	Bypass: BOOL;
	bogus: BOOL := FALSE;
	SR_FD2_new: SR;
	fbWasteBlower: TOF;
	
	bHotMeltAlarm_i:BOOL;
	
END_VAR

VAR_OUTPUT
	bHighHeatOn_i: BOOL;
	bBlowerOn_i: BOOL;
END_VAR

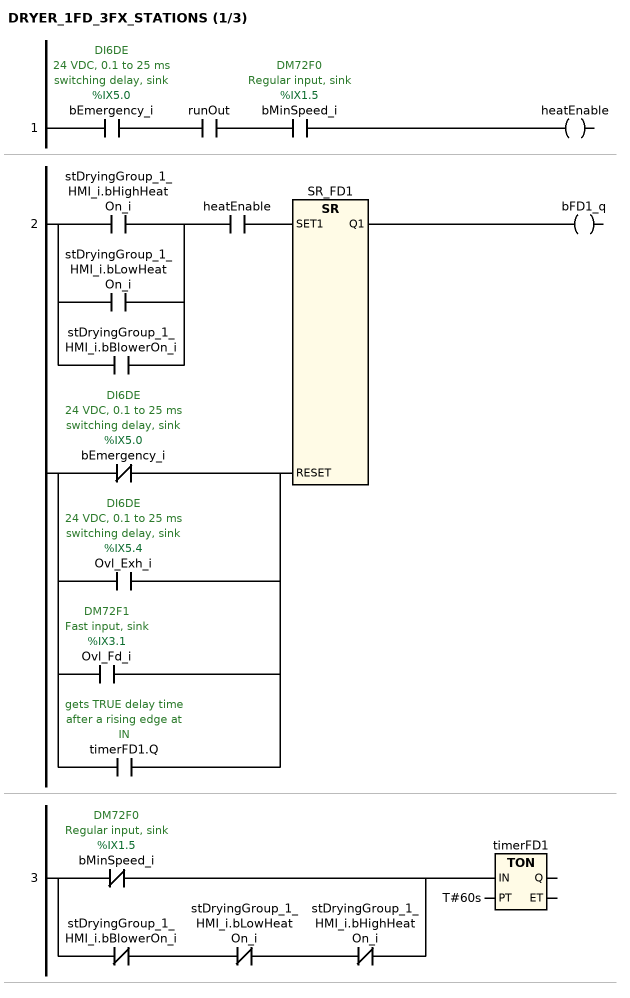
// NETWORK 1
//   bEmergency_i: DI6DE 24 VDC, 0.1 to 25 ms switching delay, sink | AT %IX5.0
//   bMinSpeed_i: DM72F0 Regular input, sink | AT %IX1.5
heatEnable := bEmergency_i AND runOut AND bMinSpeed_i;

// NETWORK 2
//   bEmergency_i: DI6DE 24 VDC, 0.1 to 25 ms switching delay, sink | AT %IX5.0
//   Ovl_Exh_i: DI6DE 24 VDC, 0.1 to 25 ms switching delay, sink | AT %IX5.4
//   Ovl_Fd_i: DM72F1 Fast input, sink | AT %IX3.1
//   timerFD1.Q: gets TRUE delay time after a rising edge at IN
SR_FD1(SET1 := (stDryingGroup_1_HMI_i.bHighHeatOn_i OR stDryingGroup_1_HMI_i.bLowHeatOn_i OR stDryingGroup_1_HMI_i.bBlowerOn_i) AND heatEnable, RESET := NOT bEmergency_i OR Ovl_Exh_i OR Ovl_Fd_i OR timerFD1.Q); // SR
bFD1_q := SR_FD1.Q1;

// NETWORK 3
//   bMinSpeed_i: DM72F0 Regular input, sink | AT %IX1.5
timerFD1(IN := NOT bMinSpeed_i OR NOT stDryingGroup_1_HMI_i.bBlowerOn_i AND NOT stDryingGroup_1_HMI_i.bLowHeatOn_i AND NOT stDryingGroup_1_HMI_i.bHighHeatOn_i, PT := T#60s); // TON

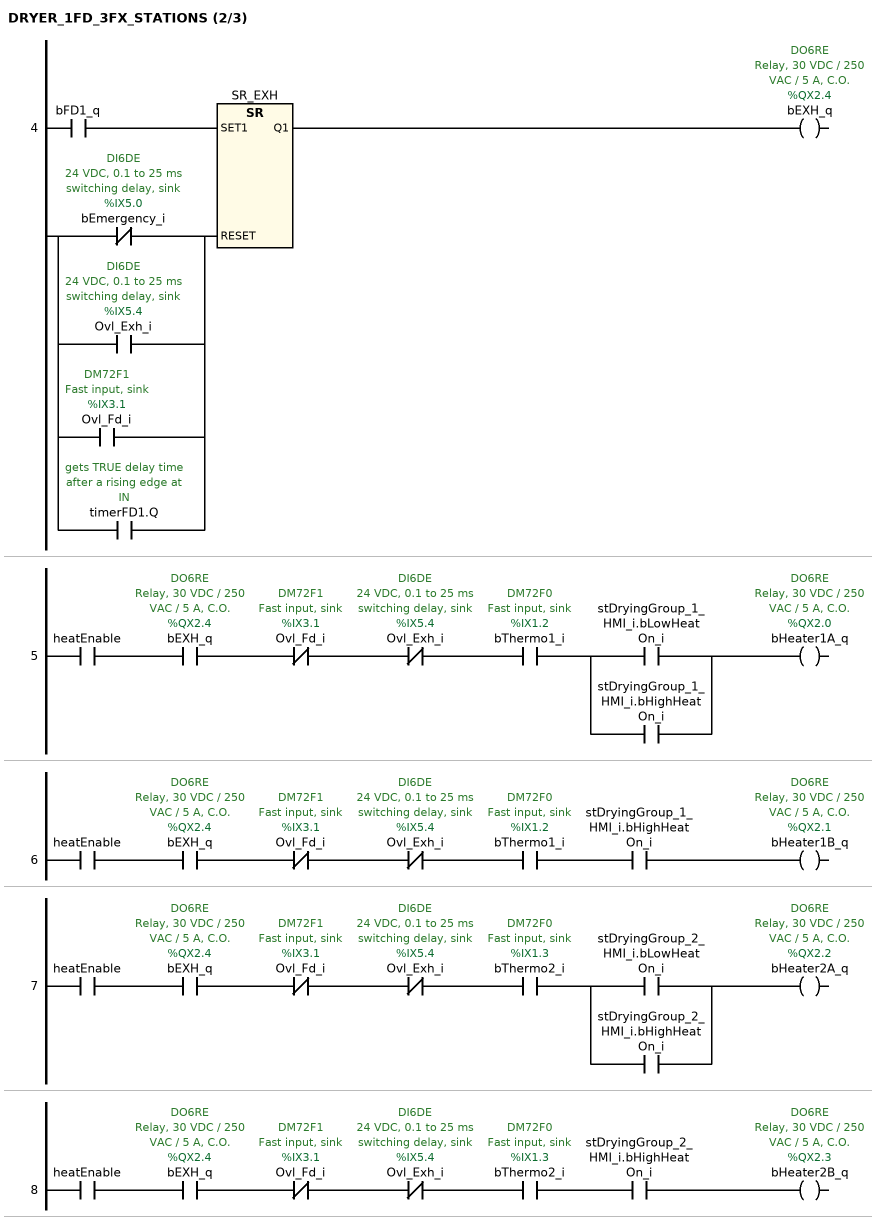
// NETWORK 4
//   bEmergency_i: DI6DE 24 VDC, 0.1 to 25 ms switching delay, sink | AT %IX5.0
//   Ovl_Exh_i: DI6DE 24 VDC, 0.1 to 25 ms switching delay, sink | AT %IX5.4
//   Ovl_Fd_i: DM72F1 Fast input, sink | AT %IX3.1
//   timerFD1.Q: gets TRUE delay time after a rising edge at IN
//   bEXH_q: DO6RE Relay, 30 VDC / 250 VAC / 5 A, C.O. | AT %QX2.4
SR_EXH(SET1 := bFD1_q, RESET := NOT bEmergency_i OR Ovl_Exh_i OR Ovl_Fd_i OR timerFD1.Q); // SR
bEXH_q := SR_EXH.Q1;

// NETWORK 5
//   bEXH_q: DO6RE Relay, 30 VDC / 250 VAC / 5 A, C.O. | AT %QX2.4
//   Ovl_Fd_i: DM72F1 Fast input, sink | AT %IX3.1
//   Ovl_Exh_i: DI6DE 24 VDC, 0.1 to 25 ms switching delay, sink | AT %IX5.4
//   bThermo1_i: DM72F0 Fast input, sink | AT %IX1.2
//   bHeater1A_q: DO6RE Relay, 30 VDC / 250 VAC / 5 A, C.O. | AT %QX2.0
bHeater1A_q := heatEnable AND bEXH_q AND NOT Ovl_Fd_i AND NOT Ovl_Exh_i AND bThermo1_i AND (stDryingGroup_1_HMI_i.bLowHeatOn_i OR stDryingGroup_1_HMI_i.bHighHeatOn_i);

// NETWORK 6
//   bEXH_q: DO6RE Relay, 30 VDC / 250 VAC / 5 A, C.O. | AT %QX2.4
//   Ovl_Fd_i: DM72F1 Fast input, sink | AT %IX3.1
//   Ovl_Exh_i: DI6DE 24 VDC, 0.1 to 25 ms switching delay, sink | AT %IX5.4
//   bThermo1_i: DM72F0 Fast input, sink | AT %IX1.2
//   bHeater1B_q: DO6RE Relay, 30 VDC / 250 VAC / 5 A, C.O. | AT %QX2.1
bHeater1B_q := heatEnable AND bEXH_q AND NOT Ovl_Fd_i AND NOT Ovl_Exh_i AND bThermo1_i AND stDryingGroup_1_HMI_i.bHighHeatOn_i;

// NETWORK 7
//   bEXH_q: DO6RE Relay, 30 VDC / 250 VAC / 5 A, C.O. | AT %QX2.4
//   Ovl_Fd_i: DM72F1 Fast input, sink | AT %IX3.1
//   Ovl_Exh_i: DI6DE 24 VDC, 0.1 to 25 ms switching delay, sink | AT %IX5.4
//   bThermo2_i: DM72F0 Fast input, sink | AT %IX1.3
//   bHeater2A_q: DO6RE Relay, 30 VDC / 250 VAC / 5 A, C.O. | AT %QX2.2
bHeater2A_q := heatEnable AND bEXH_q AND NOT Ovl_Fd_i AND NOT Ovl_Exh_i AND bThermo2_i AND (stDryingGroup_2_HMI_i.bLowHeatOn_i OR stDryingGroup_2_HMI_i.bHighHeatOn_i);

// NETWORK 8
//   bEXH_q: DO6RE Relay, 30 VDC / 250 VAC / 5 A, C.O. | AT %QX2.4
//   Ovl_Fd_i: DM72F1 Fast input, sink | AT %IX3.1
//   Ovl_Exh_i: DI6DE 24 VDC, 0.1 to 25 ms switching delay, sink | AT %IX5.4
//   bThermo2_i: DM72F0 Fast input, sink | AT %IX1.3
//   bHeater2B_q: DO6RE Relay, 30 VDC / 250 VAC / 5 A, C.O. | AT %QX2.3
bHeater2B_q := heatEnable AND bEXH_q AND NOT Ovl_Fd_i AND NOT Ovl_Exh_i AND bThermo2_i AND stDryingGroup_2_HMI_i.bHighHeatOn_i;

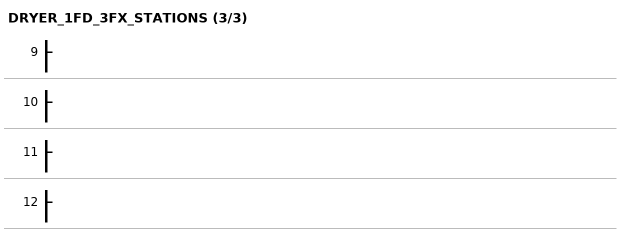
// NETWORK 9

// NETWORK 10

// NETWORK 11

// NETWORK 12

END_PROGRAM

// MyController/Application/ETH_NETWORK
PROGRAM ETH_NETWORK
VAR
	

	NewWord: WORD;
	NewBool:	BOOL;
	
	ReINIT:BOOL := FALSE;
	bTest_MinSpeed_i:BOOL := FALSE;
	
	
	FromRewind:WORD	:=	0;
	fbTP_STARTUP: TP;
	tStartUp_Time:TIME;
	AniloxModbusError2: BOOL;
	
	RexrothModbusError: BOOL;
	
	FB_RegPos: TP;
	FB_RegNeg: TP;
	
	FB_JogPos: TP;
	FB_JogNeg: TP;
END_VAR




bStartUpBit	:= TRUE;
fbTP_STARTUP(IN:=bStartUpBit , PT:= T#3S, Q=> bStartUp_ResetBit, ET=> tStartUp_Time);
fbTP_STARTUP(IN:=bStartUpBit , PT:= T#3S, Q=> bStartUp_SetBit, ET=> tStartUp_Time);

IF bStartUp_SetBit = TRUE AND uiUnwindTensManual_HMI_i = 0 THEN
	
	uiUnwindTensManual_HMI_i:= 10;
END_IF


wPar1838_PidOn_ETH.0 := bRewindPID_Out; 
InfeedModbusError	:= IoConfig_Globals.INFEED_Instance.xError;


IF InfeedModbusError = TRUE THEN

	
	IoConfig_Globals.INFEED_Instance.xConfirmError := TRUE;

ELSE		
	IoConfig_Globals.INFEED_Instance.xConfirmError := FALSE;
END_IF



RewindModbusError	:= IoConfig_Globals.REWIND_DF_Instance.xError;


IF RewindModbusError = TRUE THEN

	IoConfig_Globals.REWIND_DF_Instance.xConfirmError := TRUE;

ELSE		
	IoConfig_Globals.REWIND_DF_Instance.xConfirmError := FALSE;
END_IF


// TOP REWIND COMM ERROR MANAGE
TopRewindModbusError	:= IoConfig_Globals.TOP_REWIND_Instance.xError;

IF TopRewindModbusError = TRUE THEN

	
	IoConfig_Globals.TOP_REWIND_Instance.xConfirmError := TRUE;

ELSE		
	IoConfig_Globals.TOP_REWIND_Instance.xConfirmError := FALSE;
END_IF



// GRAVURE COMM ERROR MANAGE
GravureModbusError	:= IoConfig_Globals.GRAVURE_Instance.xError;

IF GravureModbusError = TRUE THEN

	
	IoConfig_Globals.GRAVURE_Instance.xConfirmError := TRUE;

ELSE		
	IoConfig_Globals.GRAVURE_Instance.xConfirmError := FALSE;
END_IF


IF gravureOnOut = TRUE THEN
	
//wRexrothCmd.0;
NewBool:= TRUE;
ELSE
NewBool:= FALSE;
//wRexrothCmd.0;

END_IF


//ANILOX COMM ERROR MANAGE

AniloxModbusError	:= IoConfig_Globals.ANILOX_1_Instance.xError;
//IoConfig_Globals.REWIND_Instance.xConfirmError := ReINIT;

IF AniloxModbusError = TRUE THEN

	IoConfig_Globals.ANILOX_1_Instance.xConfirmError := TRUE;

ELSE		
	IoConfig_Globals.ANILOX_1_Instance.xConfirmError := FALSE;
END_IF


AniloxModbusError2	:= IoConfig_Globals.ANILOX_2_Instance.xError;
//IoConfig_Globals.REWIND_Instance.xConfirmError := ReINIT;

IF AniloxModbusError2 = TRUE THEN

	IoConfig_Globals.ANILOX_2_Instance.xConfirmError := TRUE;

ELSE		
	IoConfig_Globals.ANILOX_2_Instance.xConfirmError := FALSE;
END_IF

IF infeedOnOut = TRUE THEN
	
	wPar1837_InfeedOn_ETH	:= 1;
ELSE
	wPar1837_InfeedOn_ETH	:= 0;

END_IF


IF bGravureRegiOn_HMI_q = TRUE THEN
	
	wPar1838_FilterOn_ETH	:= 1;
ELSE
	wPar1838_FilterOn_ETH	:= 0;

END_IF



//REWIND ON / OFF
IF (rewindOnOut = TRUE ) THEN
	
	wPar1837_RewindOn_ETH	:= 1;
ELSE
	wPar1837_RewindOn_ETH	:= 0;
	
END_IF


//REWIND PID ON
IF bRewindPID_Out = TRUE THEN
	
	wPar1838_PidOn_ETH	:= 1;
	
ELSE
	wPar1838_PidOn_ETH	:= 0;

	
END_IF



//TOP REWIND ON / OFF
IF GVL_HMI.top_rewindOnOut  = TRUE THEN
	

	wPar1837_TopRewindOn_ETH	:= 1;
ELSE
	wPar1837_TopRewindOn_ETH	:= 0;
	
END_IF


//TOP REWIND PID ON  (SAME SIGNAL)
IF bRewindPID_Out = TRUE THEN
	
	wPar1838_TopPidOn_ETH	:= 1;
	
ELSE
	wPar1838_TopPidOn_ETH	:= 0;

	
END_IF

//TOP REWIND ON / OFF
IF GVL_HMI.gravureOnOut  = TRUE THEN
	

	wPar1837_GravureOn_ETH	:= 1;
ELSE
	wPar1837_GravureOn_ETH	:= 0;
	
END_IF



IF ArFlexoStation[1].bAniloxMot_q = TRUE THEN
	
	wPar1838_ProcessOn_ETH := 0;	//ANILOX
ELSE
	wPar1838_ProcessOn_ETH := 1;	//ANILOX
END_IF

IF ArFlexoStation[2].bAniloxMot_q = TRUE THEN
	
	wPar1838_ProcessOn_2_ETH := 0;	//ANILOX
ELSE
	wPar1838_ProcessOn_2_ETH := 1;	//ANILOX
END_IF

wPar1839_AniloxFWD_ETH.0 	:= recto1Out;
wPar1840_AniloxBCK_ETH.0	:=	verso1Out;


wPar1839_AniloxFWD_2_ETH.0 	:= recto2Out;
wPar1840_AniloxBCK_2_ETH.0	:=	verso2Out;


IF (wPar2019_DryPermit_ETH.0) = TRUE THEN
	
	bTest_MinSpeed_i	:= 1;
ELSE
	bTest_MinSpeed_i	:= 0;
	
END_IF


IF (	(bArAniloxMotor_KEEP[1]) = TRUE) AND (NOT bArSETUP_KEEP[1]) THEN	


	wPar1837_AniloxOn_ETH	:= 1;
ELSE
	wPar1837_AniloxOn_ETH	:= 0;
	
END_IF


IF (	(bArAniloxMotor_KEEP[2]) = TRUE) AND (NOT bArSETUP_KEEP[2]) THEN	


	wPar1837_AniloxOn_2_ETH	:= 1;
ELSE
	wPar1837_AniloxOn_2_ETH	:= 0;
	
END_IF




IF (rollendOnOut = FALSE) THEN

	uiRollEndState := 0 ;
	
ELSIF ((rollendOnOut = TRUE) AND (bEndOfRoll_Reached = FALSE)) THEN

	uiRollEndState := 1 ;
	
ELSIF ((rollendOnOut = TRUE) AND (bEndOfRoll_Reached = TRUE)) THEN
	
	uiRollEndState := 2 ;
	
END_IF


bRewindHealthy_ETH := wPar1001_RewindHealthy_ETH.0;

bRewindActive_ETH	:= wPar1002_RewindActive_ETH.0;

bTopRewindHealthy_ETH := wPar1001_TopRewindHealthy_ETH.0;

bTopRewindActive_ETH	:= wPar1002_TopRewindActive_ETH.0;

bInfeedHealthy_ETH := 1;//wPar1001_InfeedHealthy_ETH.0;

bInfeedActive_ETH	:=  1;//wPar1002_InfeedActive_ETH.0;

IF ((bRewindHealthy_ETH AND bRewindActive_ETH) OR ( bConveyorOn_HMI_i) OR  (bTopRewindHealthy_ETH AND bTopRewindActive_ETH)) AND bInfeedHealthy_ETH AND bInfeedActive_ETH THEN
	
	bAllDrivesOK_TO_RUN_ETH := TRUE;
ELSE
	bAllDrivesOK_TO_RUN_ETH := FALSE;
	
END_IF

IF (bRewindHealthy_ETH AND bRewindActive_ETH) OR (bTopRewindHealthy_ETH AND bTopRewindActive_ETH) OR ( bConveyorOn_HMI_i) THEN

	bRewindRunSignalMissing_HMI := FALSE;
ELSE
	bRewindRunSignalMissing_HMI	:= TRUE;
END_IF

IF bInfeedHealthy_ETH AND bInfeedActive_ETH THEN

	bInfeedRunSignalMissing_HMI := FALSE;
ELSE
	bInfeedRunSignalMissing_HMI	:= TRUE;
END_IF


IF InfeedModbusError = TRUE OR RewindModbusError = TRUE  THEN
	
	bAllDrives_ModbusError_HMI := TRUE;
ELSE
	bAllDrives_ModbusError_HMI := FALSE;

END_IF

//****************************************
//*** GRAVURE COMMUNICATION MANAGEMENT ***
//****************************************

IoConfig_Globals.REXROTH_1_Instance.xBusy;
IoConfig_Globals.REXROTH_1_Instance.xError;
IoConfig_Globals.REXROTH_1_Instance.xDone;

// GRAVURE COMM ERROR MANAGE
RexrothModbusError	:= IoConfig_Globals.REXROTH_1_Instance.xError;

IF RexrothModbusError = TRUE THEN

	IoConfig_Globals.REXROTH_1_Instance.xConfirmError 	:= TRUE;
	
ELSE

	IoConfig_Globals.REXROTH_1_Instance.xConfirmError 	:= FALSE;

END_IF

	//IoConfig_Globals.REXROTH_1_Instance.x


bCounterReached_HMI_q := wPar1933_CountReach_ETH.0;

bGravure_Tens_Inc_ETH_q	:= bGravure_Tens_Inc_HMI_i;
bGravure_Tens_Dec_ETH_q	:= bGravure_Tens_Dec_HMI_i;
//bGravure_Tens_Inc_i	:= bGravure_Tens_Inc_HMI_i;
//bGravure_Tens_Dec_i	:= bGravure_Tens_Dec_HMI_i;
FB_RegPos(IN:=bGravure_Reg_Adv_HMI_i OR ArFlexoStation[1].bRegAdvance_q , PT:=T#250MS , Q=> , ET=> );
FB_RegNeg(IN:=bGravure_Reg_Ret_HMI_i OR ArFlexoStation[1].bRegRetard_q , PT:=T#250MS , Q=> , ET=> );

	bGravure_Reg_Adv_ETH_q	:= FB_RegPos.Q;
	bGravure_Reg_Ret_ETH_q	:= FB_RegNeg.Q;
	bGravureOn_ETH_q		:=	gravureOnOut;

	
	bGravureRegiOn_HMI_q		:=	bGravure_RegiCtrlOn_HMI_i;
	bInfeedRegiOn_HMI_q			:=	bInfeed_RegiCtrlOn_HMI_i;
	
FB_JogPos(IN:=bGravure_Jog_Adv_HMI_i , PT:=T#250MS , Q=> , ET=> );
FB_JogNeg(IN:=bGravure_Jog_Ret_HMI_i , PT:=T#250MS , Q=> , ET=> );

	bGravure_Jog_Adv_HMI_q		:=	FB_JogPos.Q;
	bGravure_Jog_Ret_HMI_q		:=	FB_JogNeg.Q;
	
//uiGravureRegisterOffset := WORD_TO_UINT(wGravureRegisterOffset);
uiGravureGearingAdjust := WORD_TO_UINT(wGravureGearingAdjust);

bInfeed_Tens_Inc_ETH_i := bInfeed_Tens_Inc_HMI_i;
bInfeed_Tens_dec_ETH_i :=bInfeed_Tens_dec_HMI_i;
bInfeed_Manual_ETH_i := bInfeed_Manual_i;
bInfeed_StatusError_HMI_q := bInfeed_StatusError_ETH_q;
bInfeed_StatusDisabled_q := ( NOT(bInfeed_StatusError_ETH_q) AND NOT  (bInfeed_StatusSynch_ETH_q) AND NOT  (bInfeed_StatusSlowRot_ETH_q));
bInfeed_StatusSynch_HMI_q :=bInfeed_StatusSynch_ETH_q;
bInfeed_ResetDrive_ETH_i := bInfeed_ResetDrive_HMI_i;

END_PROGRAM

// MyController/Application/FAULT_INTERLOCK
PROGRAM FAULT_INTERLOCK
VAR
	bogus: BOOL;
	SR_AniloxOn:		SR;
	bMachineHealthy:BOOL;
	
	
	infeedOnOut_L:BOOL;
	rewindOnOut_L:BOOL;
	
	bBYPASS:BOOL:= TRUE;
	
	okToRunV2:BOOL;
	okToJogV2:BOOL;
	fbTOF_RUN: TOF;
	etRun: TIME;
	bReadyToRun: BOOL;
	bSensorsOk: BOOL;
	SR_SlowRotation: SR;
	COUNTER_REACHED: BOOL;
END_VAR
VAR // added by the converter: edge detectors and wires of the graphical bodies
    _rt1, _rt2, _rt3, _rt4, _rt5, _rt6, _rt7, _rt8, _rt9, _rt10, _rt11, _rt12 : R_TRIG;
END_VAR

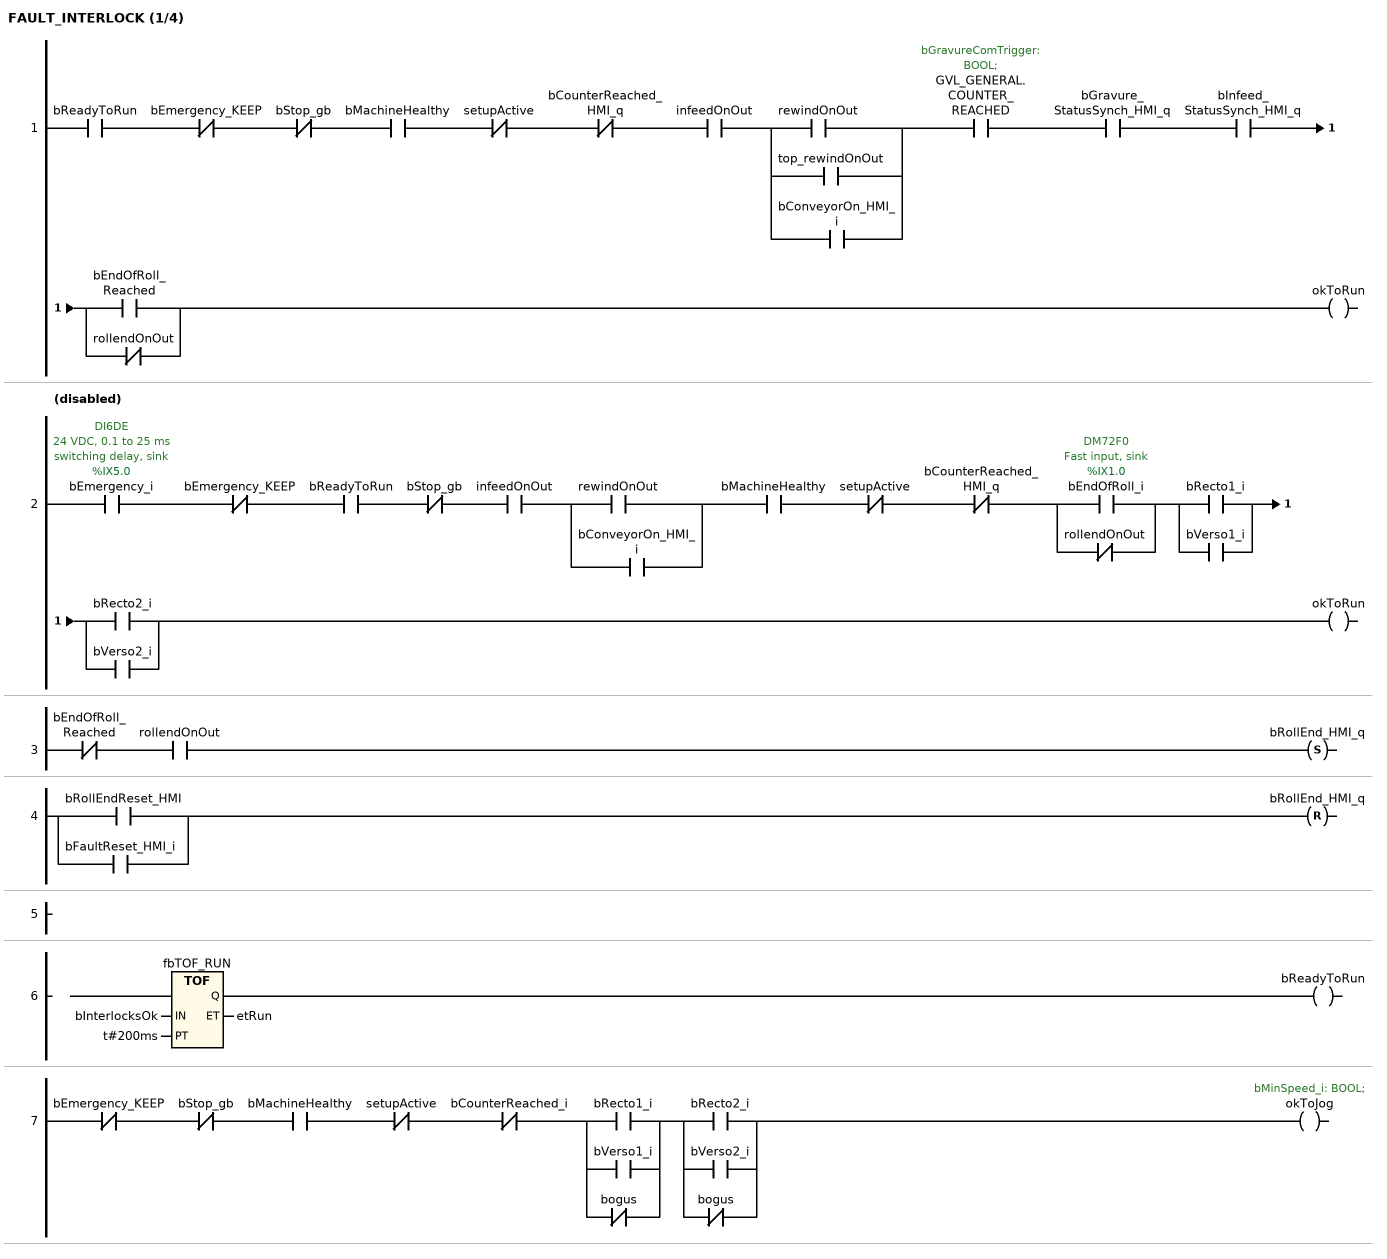
// NETWORK 1
//   GVL_GENERAL.COUNTER_REACHED: bGravureComTrigger: BOOL;
okToRun := bReadyToRun AND NOT bEmergency_KEEP AND NOT bStop_gb AND bMachineHealthy AND NOT setupActive AND NOT bCounterReached_HMI_q AND infeedOnOut AND (rewindOnOut OR top_rewindOnOut OR bConveyorOn_HMI_i) AND GVL_GENERAL.COUNTER_REACHED AND bGravure_StatusSynch_HMI_q AND bInfeed_StatusSynch_HMI_q AND (bEndOfRoll_Reached OR NOT rollendOnOut);

// NETWORK 2 (disabled)
//   bEmergency_i: DI6DE 24 VDC, 0.1 to 25 ms switching delay, sink | AT %IX5.0
//   bEndOfRoll_i: DM72F0 Fast input, sink | AT %IX1.0
// okToRun := bEmergency_i AND NOT bEmergency_KEEP AND bReadyToRun AND NOT bStop_gb AND infeedOnOut AND (rewindOnOut OR bConveyorOn_HMI_i) AND bMachineHealthy AND NOT setupActive AND NOT bCounterReached_HMI_q AND (bEndOfRoll_i OR NOT rollendOnOut) AND (bRecto1_i OR bVerso1_i) AND (bRecto2_i OR bVerso2_i);

// NETWORK 3
bRollEnd_HMI_q S= NOT bEndOfRoll_Reached AND rollendOnOut;

// NETWORK 4
bRollEnd_HMI_q R= bRollEndReset_HMI OR bFaultReset_HMI_i;

// NETWORK 5

// NETWORK 6
fbTOF_RUN(IN := bInterlocksOk, PT := t#200ms, ET => etRun); // TOF
bReadyToRun := fbTOF_RUN.Q;

// NETWORK 7
//   okToJog: bMinSpeed_i: BOOL;
okToJog := NOT bEmergency_KEEP AND NOT bStop_gb AND bMachineHealthy AND NOT setupActive AND NOT bCounterReached_i AND (bRecto1_i OR bVerso1_i OR NOT bogus) AND (bRecto2_i OR bVerso2_i OR NOT bogus);

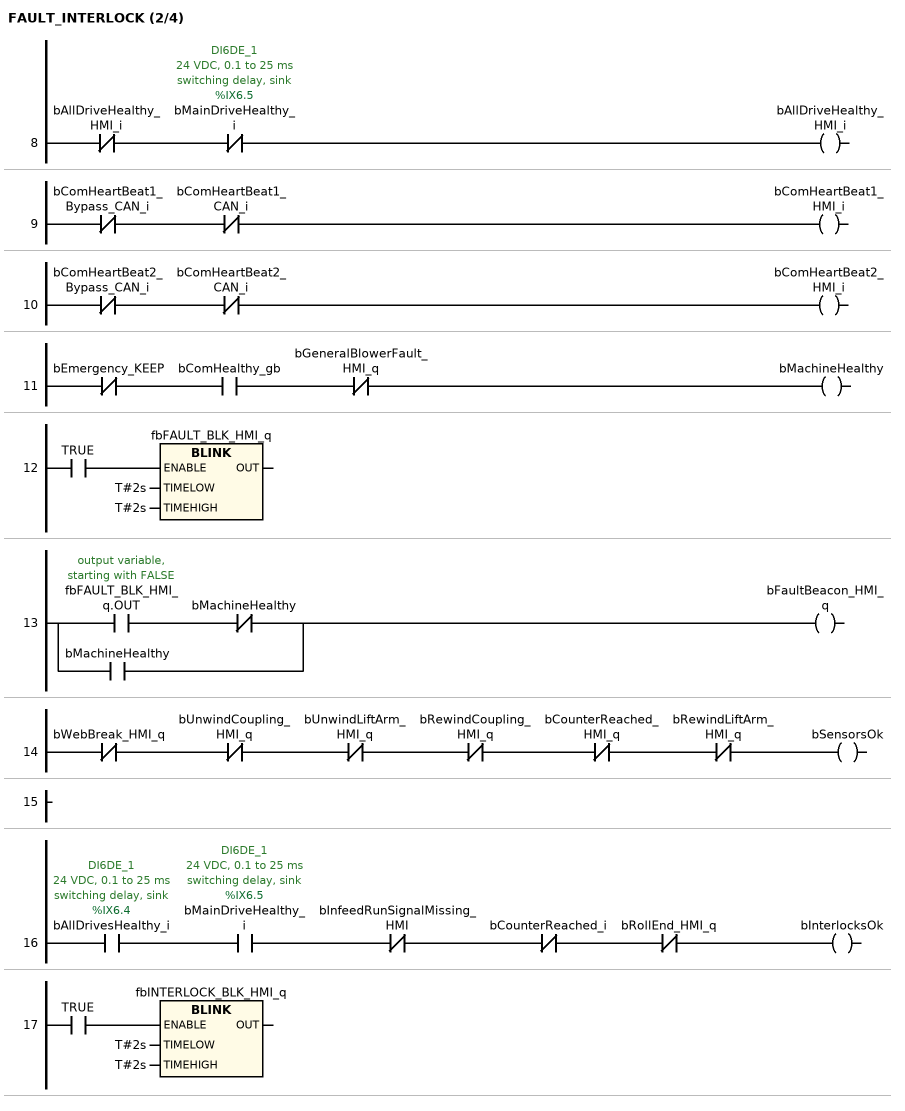
// NETWORK 8
//   bMainDriveHealthy_i: DI6DE_1 24 VDC, 0.1 to 25 ms switching delay, sink | AT %IX6.5
bAllDriveHealthy_HMI_i := NOT bAllDriveHealthy_HMI_i AND NOT bMainDriveHealthy_i;

// NETWORK 9
bComHeartBeat1_HMI_i := NOT bComHeartBeat1_Bypass_CAN_i AND NOT bComHeartBeat1_CAN_i;

// NETWORK 10
bComHeartBeat2_HMI_i := NOT bComHeartBeat2_Bypass_CAN_i AND NOT bComHeartBeat2_CAN_i;

// NETWORK 11
bMachineHealthy := NOT bEmergency_KEEP AND bComHealthy_gb AND NOT bGeneralBlowerFault_HMI_q;

// NETWORK 12
fbFAULT_BLK_HMI_q(ENABLE := TRUE, TIMELOW := T#2s, TIMEHIGH := T#2s); // BLINK

// NETWORK 13
//   fbFAULT_BLK_HMI_q.OUT: output variable, starting with FALSE
bFaultBeacon_HMI_q := fbFAULT_BLK_HMI_q.OUT AND NOT bMachineHealthy OR bMachineHealthy;

// NETWORK 14
bSensorsOk := NOT bWebBreak_HMI_q AND NOT bUnwindCoupling_HMI_q AND NOT bUnwindLiftArm_HMI_q AND NOT bRewindCoupling_HMI_q AND NOT bCounterReached_HMI_q AND NOT bRewindLiftArm_HMI_q;

// NETWORK 15

// NETWORK 16
//   bAllDrivesHealthy_i: DI6DE_1 24 VDC, 0.1 to 25 ms switching delay, sink | AT %IX6.4
//   bMainDriveHealthy_i: DI6DE_1 24 VDC, 0.1 to 25 ms switching delay, sink | AT %IX6.5
bInterlocksOk := bAllDrivesHealthy_i AND bMainDriveHealthy_i AND NOT bInfeedRunSignalMissing_HMI AND NOT bCounterReached_i AND NOT bRollEnd_HMI_q;

// NETWORK 17
fbINTERLOCK_BLK_HMI_q(ENABLE := TRUE, TIMELOW := T#2s, TIMEHIGH := T#2s); // BLINK

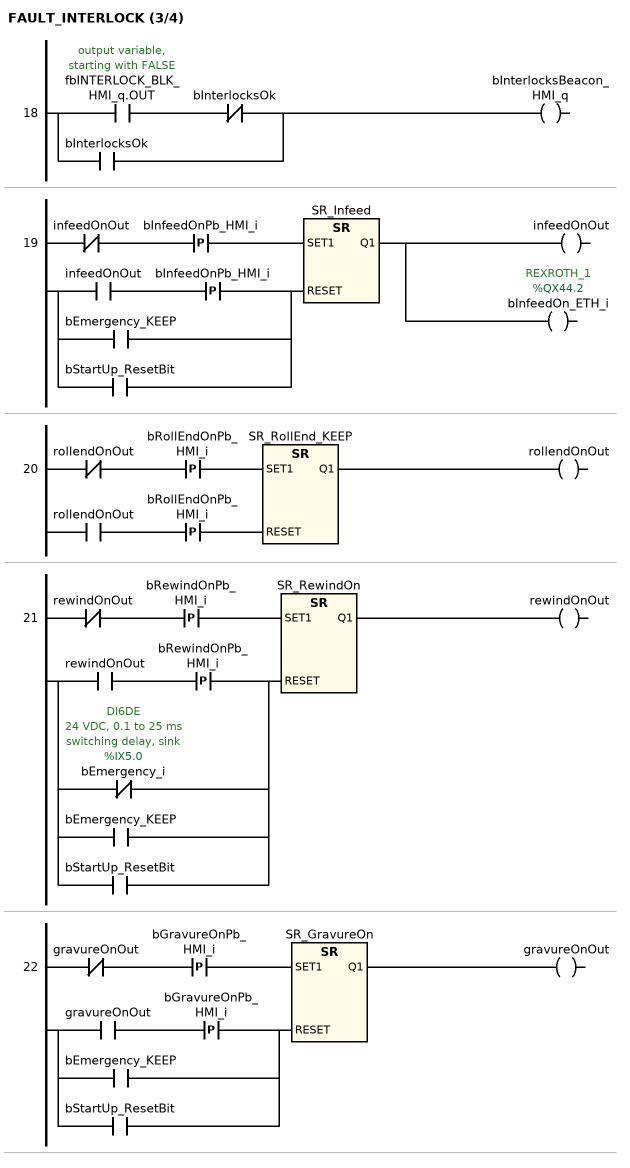
// NETWORK 18
//   fbINTERLOCK_BLK_HMI_q.OUT: output variable, starting with FALSE
bInterlocksBeacon_HMI_q := fbINTERLOCK_BLK_HMI_q.OUT AND NOT bInterlocksOk OR bInterlocksOk;

// NETWORK 19
//   bInfeedOn_ETH_i: REXROTH_1 | AT %QX44.2
_rt1(CLK := bInfeedOnPb_HMI_i);
_rt2(CLK := bInfeedOnPb_HMI_i);
SR_Infeed(SET1 := NOT infeedOnOut AND _rt1.Q, RESET := infeedOnOut AND _rt2.Q OR bEmergency_KEEP OR bStartUp_ResetBit); // SR
infeedOnOut := SR_Infeed.Q1;
bInfeedOn_ETH_i := SR_Infeed.Q1;

// NETWORK 20
//   SR_RollEnd_KEEP: bIR1_KEEP:BOOL := FALSE; bIR2_KEEP:BOOL := FALSE; bIR3_KEEP:BOOL := FALSE; bIR4_KEEP:BOOL := FALSE;
_rt3(CLK := bRollEndOnPb_HMI_i);
_rt4(CLK := bRollEndOnPb_HMI_i);
SR_RollEnd_KEEP(SET1 := NOT rollendOnOut AND _rt3.Q, RESET := rollendOnOut AND _rt4.Q); // SR
rollendOnOut := SR_RollEnd_KEEP.Q1;

// NETWORK 21
//   bEmergency_i: DI6DE 24 VDC, 0.1 to 25 ms switching delay, sink | AT %IX5.0
_rt5(CLK := bRewindOnPb_HMI_i);
_rt6(CLK := bRewindOnPb_HMI_i);
SR_RewindOn(SET1 := NOT rewindOnOut AND _rt5.Q, RESET := rewindOnOut AND _rt6.Q OR NOT bEmergency_i OR bEmergency_KEEP OR bStartUp_ResetBit); // SR
rewindOnOut := SR_RewindOn.Q1;

// NETWORK 22
_rt7(CLK := bGravureOnPb_HMI_i);
_rt8(CLK := bGravureOnPb_HMI_i);
SR_GravureOn(SET1 := NOT gravureOnOut AND _rt7.Q, RESET := gravureOnOut AND _rt8.Q OR bEmergency_KEEP OR bStartUp_ResetBit); // SR
gravureOnOut := SR_GravureOn.Q1;

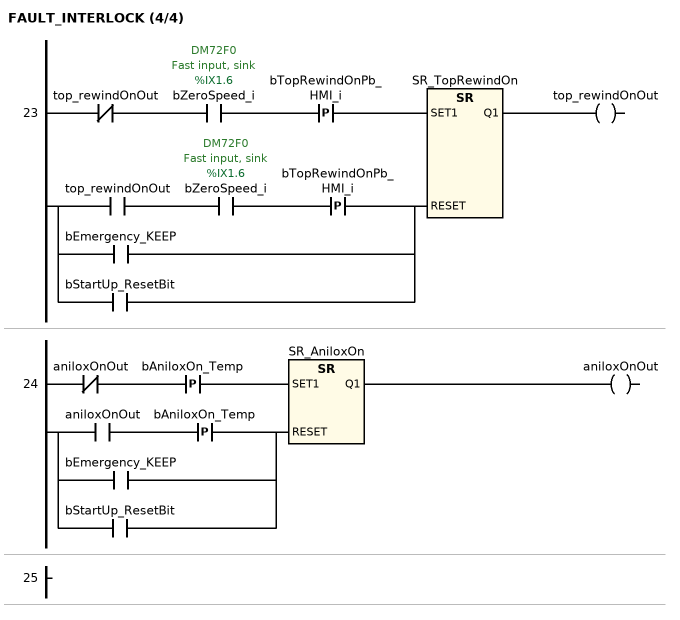
// NETWORK 23
//   bZeroSpeed_i: DM72F0 Fast input, sink | AT %IX1.6
_rt9(CLK := bTopRewindOnPb_HMI_i);
_rt10(CLK := bTopRewindOnPb_HMI_i);
SR_TopRewindOn(SET1 := NOT top_rewindOnOut AND bZeroSpeed_i AND _rt9.Q, RESET := top_rewindOnOut AND bZeroSpeed_i AND _rt10.Q OR bEmergency_KEEP OR bStartUp_ResetBit); // SR
top_rewindOnOut := SR_TopRewindOn.Q1;

// NETWORK 24
_rt11(CLK := bAniloxOn_Temp);
_rt12(CLK := bAniloxOn_Temp);
SR_AniloxOn(SET1 := NOT aniloxOnOut AND _rt11.Q, RESET := aniloxOnOut AND _rt12.Q OR bEmergency_KEEP OR bStartUp_ResetBit); // SR
aniloxOnOut := SR_AniloxOn.Q1;

// NETWORK 25

END_PROGRAM

// MyController/Application/GRAVURE_PGM
PROGRAM GRAVURE_PGM
VAR
	FB_Gravure_Kickoff: SR;
	bEnableGravureCom:BOOL	:= TRUE;
	fbCOM_TRIGGER:BLINK;
	SR_SlowRotation:SR;

	
END_VAR
VAR // added by the converter: edge detectors and wires of the graphical bodies
    _rt1, _rt2, _rt3, _rt4 : R_TRIG;
    _w1 : BOOL;
END_VAR

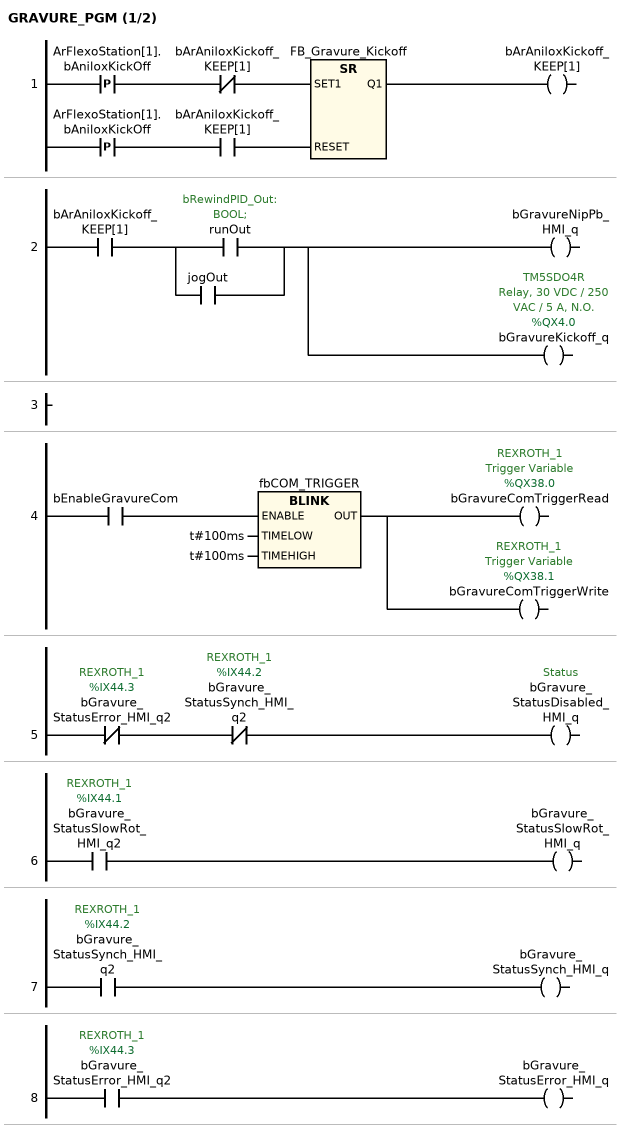
// NETWORK 1
_rt1(CLK := ArFlexoStation[1].bAniloxKickOff);
_rt2(CLK := ArFlexoStation[1].bAniloxKickOff);
FB_Gravure_Kickoff(SET1 := _rt1.Q AND NOT bArAniloxKickoff_KEEP[1], RESET := _rt2.Q AND bArAniloxKickoff_KEEP[1]); // SR
bArAniloxKickoff_KEEP[1] := FB_Gravure_Kickoff.Q1;

// NETWORK 2
//   runOut: bRewindPID_Out:BOOL;
//   bGravureKickoff_q: TM5SDO4R Relay, 30 VDC / 250 VAC / 5 A, N.O. | AT %QX4.0
_w1 := bArAniloxKickoff_KEEP[1] AND (runOut OR jogOut);
bGravureNipPb_HMI_q := _w1;
bGravureKickoff_q := _w1;

// NETWORK 3

// NETWORK 4
//   bGravureComTriggerRead: REXROTH_1 Trigger Variable | AT %QX38.0
//   bGravureComTriggerWrite: REXROTH_1 Trigger Variable | AT %QX38.1
fbCOM_TRIGGER(ENABLE := bEnableGravureCom, TIMELOW := t#100ms, TIMEHIGH := t#100ms); // BLINK
bGravureComTriggerRead := fbCOM_TRIGGER.OUT;
bGravureComTriggerWrite := fbCOM_TRIGGER.OUT;

// NETWORK 5
//   bGravure_StatusError_HMI_q2: REXROTH_1 | AT %IX44.3
//   bGravure_StatusSynch_HMI_q2: REXROTH_1 | AT %IX44.2
//   bGravure_StatusDisabled_HMI_q: Status
bGravure_StatusDisabled_HMI_q := NOT bGravure_StatusError_HMI_q2 AND NOT bGravure_StatusSynch_HMI_q2;

// NETWORK 6
//   bGravure_StatusSlowRot_HMI_q2: REXROTH_1 | AT %IX44.1
bGravure_StatusSlowRot_HMI_q := bGravure_StatusSlowRot_HMI_q2;

// NETWORK 7
//   bGravure_StatusSynch_HMI_q2: REXROTH_1 | AT %IX44.2
bGravure_StatusSynch_HMI_q := bGravure_StatusSynch_HMI_q2;

// NETWORK 8
//   bGravure_StatusError_HMI_q2: REXROTH_1 | AT %IX44.3
bGravure_StatusError_HMI_q := bGravure_StatusError_HMI_q2;

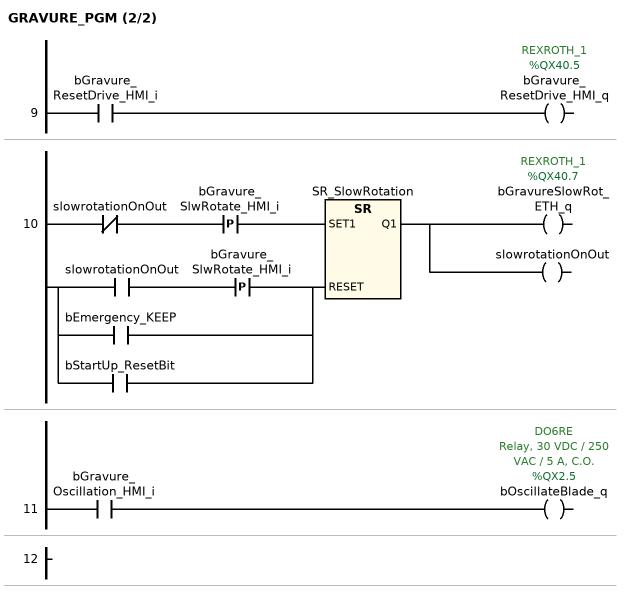
// NETWORK 9
//   bGravure_ResetDrive_HMI_q: REXROTH_1 | AT %QX40.5
bGravure_ResetDrive_HMI_q := bGravure_ResetDrive_HMI_i;

// NETWORK 10
//   bGravureSlowRot_ETH_q: REXROTH_1 | AT %QX40.7
_rt3(CLK := bGravure_SlwRotate_HMI_i);
_rt4(CLK := bGravure_SlwRotate_HMI_i);
SR_SlowRotation(SET1 := NOT slowrotationOnOut AND _rt3.Q, RESET := slowrotationOnOut AND _rt4.Q OR bEmergency_KEEP OR bStartUp_ResetBit); // SR
bGravureSlowRot_ETH_q := SR_SlowRotation.Q1;
slowrotationOnOut := SR_SlowRotation.Q1;

// NETWORK 11
//   bOscillateBlade_q: DO6RE Relay, 30 VDC / 250 VAC / 5 A, C.O. | AT %QX2.5
bOscillateBlade_q := bGravure_Oscillation_HMI_i;

// NETWORK 12

END_PROGRAM

// MyController/Application/LATCH_ERROR
PROGRAM LATCH_ERROR

VAR


	fbF_TRIG1: F_TRIG;
	SR_CAN_COMM: SR;
	SR_ETH_COMM: SR;
	fbR_TRIG2: R_TRIG;
	SR_GBX1: SR;
	fbR_TRIG3: F_TRIG;
	fbR_TRIG4: F_TRIG;
	SR_GBX2: SR;
	SR_InfeedRunSignalMissing: SR;
	SR_RewindRunSignalMissing: SR;
	fbR_TRIG5: F_TRIG;
	fbR_TRIG6: F_TRIG;
	fbF_TRIG5: F_TRIG;
	fbF_TRIG6: F_TRIG;
	bInfeed_Error: BOOL;
	bRewind_Error: BOOL;
	
	bRewindCoupling_Error: BOOL;
	SR_UnwindCoupling: SR;
	SR_UnwindLiftArm: SR;
	
	SR_RewindCoupling: SR;
	SR_RewindLiftArm: SR;
	SR_SafetyGuard: SR;
	SR_WebBreak: SR;
	SR_ExhaustOVL: SR;
	SR_EnableRewindLift: SR;
	SR_Emergency2: SR;
	SR_AllDrivesOK_ETH: SR;
	bAllDrivesOK_ETH_FAULT: BOOL;
	SR_MODBUS_Error: SR;
	bModbusTCP_Error: BOOL;
	bInterlock_Error: BOOL;
	SR_INTERLOCK_Error: SR;
	
	
	//Modif Antoine->Gravure
	SR_Gravure: SR;
	b_Gravure_i: BOOL := false;
	b_Gravure_q: BOOL := FALSE;	//K1
END_VAR
VAR // added by the converter: edge detectors and wires of the graphical bodies
    _rt1, _rt2, _rt3, _rt4, _rt5, _rt6, _rt7, _rt8, _rt9, _rt10, _rt11, _rt12, _rt13, _rt14, _rt15, _rt16 : R_TRIG;
    _ft1, _ft2 : F_TRIG;
END_VAR

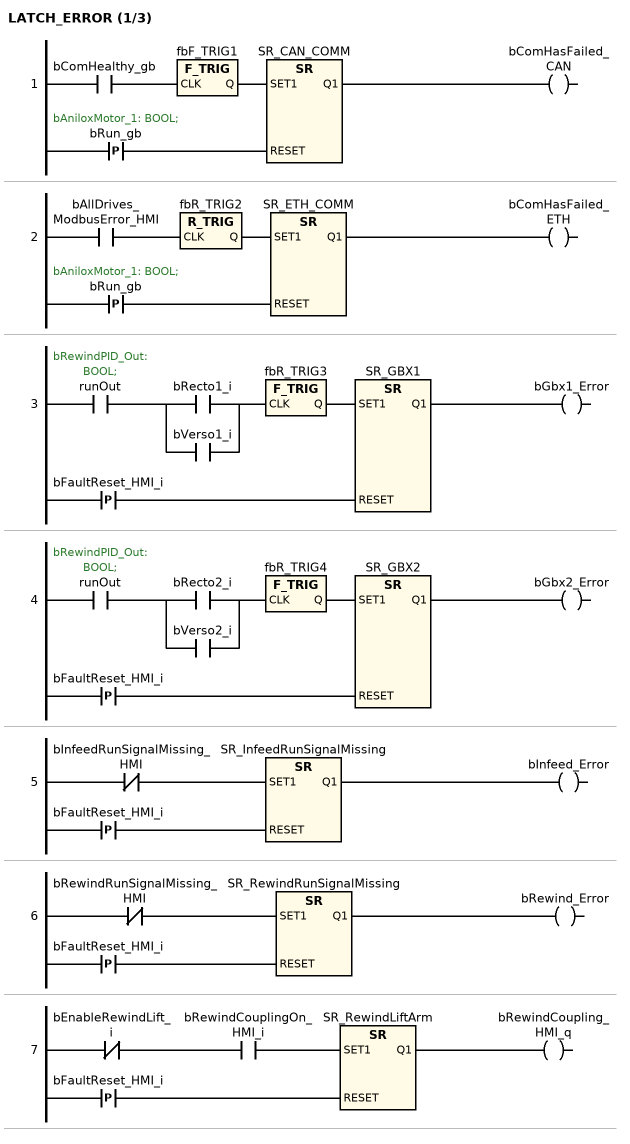
// NETWORK 1
//   bRun_gb: bAniloxMotor_1: BOOL;
fbF_TRIG1(CLK := bComHealthy_gb); // F_TRIG
_rt1(CLK := bRun_gb);
SR_CAN_COMM(SET1 := fbF_TRIG1.Q, RESET := _rt1.Q); // SR
bComHasFailed_CAN := SR_CAN_COMM.Q1;

// NETWORK 2
//   bRun_gb: bAniloxMotor_1: BOOL;
fbR_TRIG2(CLK := bAllDrives_ModbusError_HMI); // R_TRIG
_rt2(CLK := bRun_gb);
SR_ETH_COMM(SET1 := fbR_TRIG2.Q, RESET := _rt2.Q); // SR
bComHasFailed_ETH := SR_ETH_COMM.Q1;

// NETWORK 3
//   runOut: bRewindPID_Out:BOOL;
fbR_TRIG3(CLK := runOut AND (bRecto1_i OR bVerso1_i)); // F_TRIG
_rt3(CLK := bFaultReset_HMI_i);
SR_GBX1(SET1 := fbR_TRIG3.Q, RESET := _rt3.Q); // SR
bGbx1_Error := SR_GBX1.Q1;

// NETWORK 4
//   runOut: bRewindPID_Out:BOOL;
fbR_TRIG4(CLK := runOut AND (bRecto2_i OR bVerso2_i)); // F_TRIG
_rt4(CLK := bFaultReset_HMI_i);
SR_GBX2(SET1 := fbR_TRIG4.Q, RESET := _rt4.Q); // SR
bGbx2_Error := SR_GBX2.Q1;

// NETWORK 5
_rt5(CLK := bFaultReset_HMI_i);
SR_InfeedRunSignalMissing(SET1 := NOT bInfeedRunSignalMissing_HMI, RESET := _rt5.Q); // SR
bInfeed_Error := SR_InfeedRunSignalMissing.Q1;

// NETWORK 6
_rt6(CLK := bFaultReset_HMI_i);
SR_RewindRunSignalMissing(SET1 := NOT bRewindRunSignalMissing_HMI, RESET := _rt6.Q); // SR
bRewind_Error := SR_RewindRunSignalMissing.Q1;

// NETWORK 7
_rt7(CLK := bFaultReset_HMI_i);
SR_RewindLiftArm(SET1 := NOT bEnableRewindLift_i AND bRewindCouplingOn_HMI_i, RESET := _rt7.Q); // SR
bRewindCoupling_HMI_q := SR_RewindLiftArm.Q1;

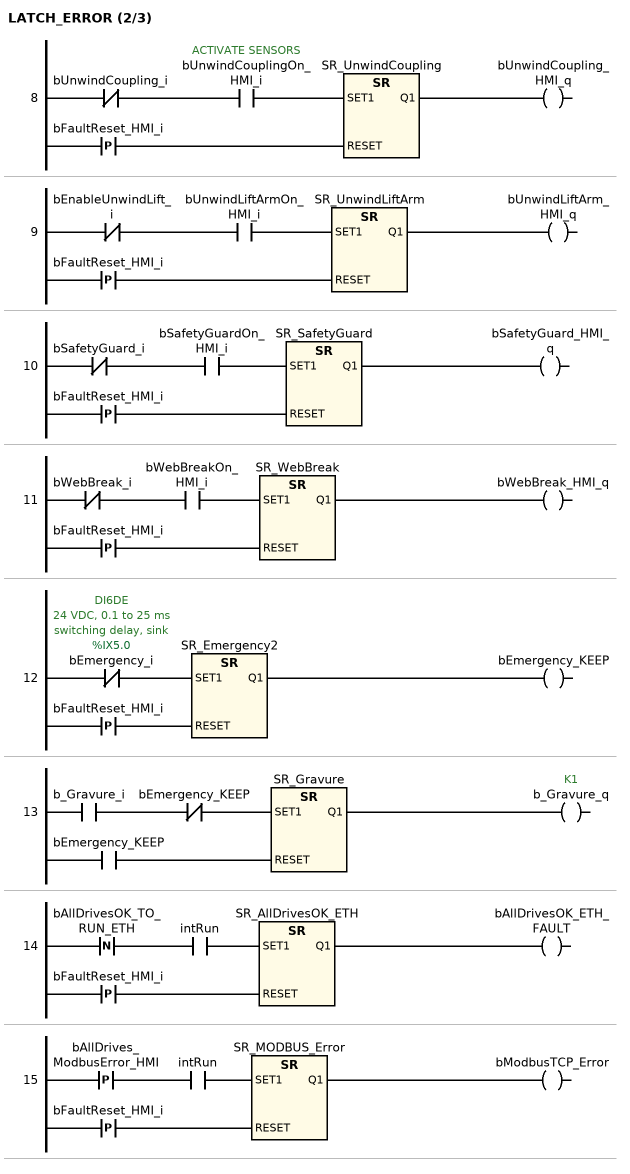
// NETWORK 8
//   bUnwindCouplingOn_HMI_i: ACTIVATE SENSORS
_rt8(CLK := bFaultReset_HMI_i);
SR_UnwindCoupling(SET1 := NOT bUnwindCoupling_i AND bUnwindCouplingOn_HMI_i, RESET := _rt8.Q); // SR
bUnwindCoupling_HMI_q := SR_UnwindCoupling.Q1;

// NETWORK 9
_rt9(CLK := bFaultReset_HMI_i);
SR_UnwindLiftArm(SET1 := NOT bEnableUnwindLift_i AND bUnwindLiftArmOn_HMI_i, RESET := _rt9.Q); // SR
bUnwindLiftArm_HMI_q := SR_UnwindLiftArm.Q1;

// NETWORK 10
_rt10(CLK := bFaultReset_HMI_i);
SR_SafetyGuard(SET1 := NOT bSafetyGuard_i AND bSafetyGuardOn_HMI_i, RESET := _rt10.Q); // SR
bSafetyGuard_HMI_q := SR_SafetyGuard.Q1;

// NETWORK 11
_rt11(CLK := bFaultReset_HMI_i);
SR_WebBreak(SET1 := NOT bWebBreak_i AND bWebBreakOn_HMI_i, RESET := _rt11.Q); // SR
bWebBreak_HMI_q := SR_WebBreak.Q1;

// NETWORK 12
//   bEmergency_i: DI6DE 24 VDC, 0.1 to 25 ms switching delay, sink | AT %IX5.0
_rt12(CLK := bFaultReset_HMI_i);
SR_Emergency2(SET1 := NOT bEmergency_i, RESET := _rt12.Q); // SR
bEmergency_KEEP := SR_Emergency2.Q1;

// NETWORK 13
//   SR_Gravure: Modif Antoine->Gravure
//   b_Gravure_q: K1
SR_Gravure(SET1 := b_Gravure_i AND NOT bEmergency_KEEP, RESET := bEmergency_KEEP); // SR
b_Gravure_q := SR_Gravure.Q1;

// NETWORK 14
_ft1(CLK := bAllDrivesOK_TO_RUN_ETH);
_rt13(CLK := bFaultReset_HMI_i);
SR_AllDrivesOK_ETH(SET1 := _ft1.Q AND intRun, RESET := _rt13.Q); // SR
bAllDrivesOK_ETH_FAULT := SR_AllDrivesOK_ETH.Q1;

// NETWORK 15
_rt14(CLK := bAllDrives_ModbusError_HMI);
_rt15(CLK := bFaultReset_HMI_i);
SR_MODBUS_Error(SET1 := _rt14.Q AND intRun, RESET := _rt15.Q); // SR
bModbusTCP_Error := SR_MODBUS_Error.Q1;

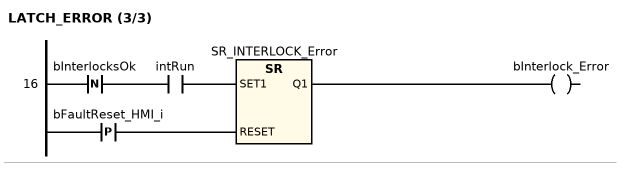
// NETWORK 16
_ft2(CLK := bInterlocksOk);
_rt16(CLK := bFaultReset_HMI_i);
SR_INTERLOCK_Error(SET1 := _ft2.Q AND intRun, RESET := _rt16.Q); // SR
bInterlock_Error := SR_INTERLOCK_Error.Q1;

END_PROGRAM

// MyController/Application/UNWIND/UNWIND_TENS_CTRL
PROGRAM UNWIND_TENS_CTRL
VAR
	fbUnwindTensCtrl: FB_PI;
	rUnwindTensionActual:REAL;
	rUnwindTensionSetpoint:REAL;
	rPID_PTERM:REAL:= 0.1;
	rPID_ITERM:REAL:= 1.0;
	bPID_HOLD: BOOL := FALSE;
	//stPID: stPiPara	:= ( Start:=[3,3], Point1 =[5,2], Point2:=[7,3], Point3:=[8,5], Point4:=[5,7], End := [3,5]); 
	stPID:stPiPara:=(tCyclTime:=T#20MS,xEnArw:=TRUE,tTn:=T#20MS,rKp:=0.06,rMaxLim:=32767.0,rMinLim:=0.0);
	bPID_ERROR:BOOL;
	
	bPID_ManualOn:BOOL;
	rPID_ManualValue:REAL:= 100.0;
	bPID_EnableStatus:BOOL;
	bPID_BusyStatus:BOOL;
	rPID_Output:REAL;
	bStatus1:BOOL;
	bError_q:BOOL;
	uiErrID:UINT;
	
	uiUnwindTensActScaled:UINT;
	diBuffer:DINT;
	bManualMode:BOOL;
	bPID_ManualModeActive:BOOL;
	uiPID_Output:UINT;
	(*OLD*)
	//uiPID_Output_q:UINT;
	rANSWER_gb:REAL;
	rStaticDemand: REAL;
	fbFilterTensOutput: Filter_MovingAverage;
	rUnwindTensionActual_HMI_q: REAL;
	rUnwindTens:REAL;
	uiSmplCnt: UINT:=99;	//HUBERT COMMENT ON JULY 8th 2014
							//Invalid parameter such as i_uiSmplCnt > 100 results in detected error and
							//corresponding detected error ID is generated.
							//During the detected error state, the output is set to zero.
							//Detected error can be reset only through the rising edge of i_xErrRst
	rPID_Output_LIM:REAL;
	abc: BOOL;
	test: UINT;
	timer25: TP;
	bFilterReset: BOOL;
	var1: real;
END_VAR
VAR // added by the converter: edge detectors and wires of the graphical bodies
    _w1, _w2, _w3, _w4, _w6, _w9, _w11, _w12 : ANY;
    _w5 : BOOL;
    _w7, _w8, _w10 : REAL;
END_VAR

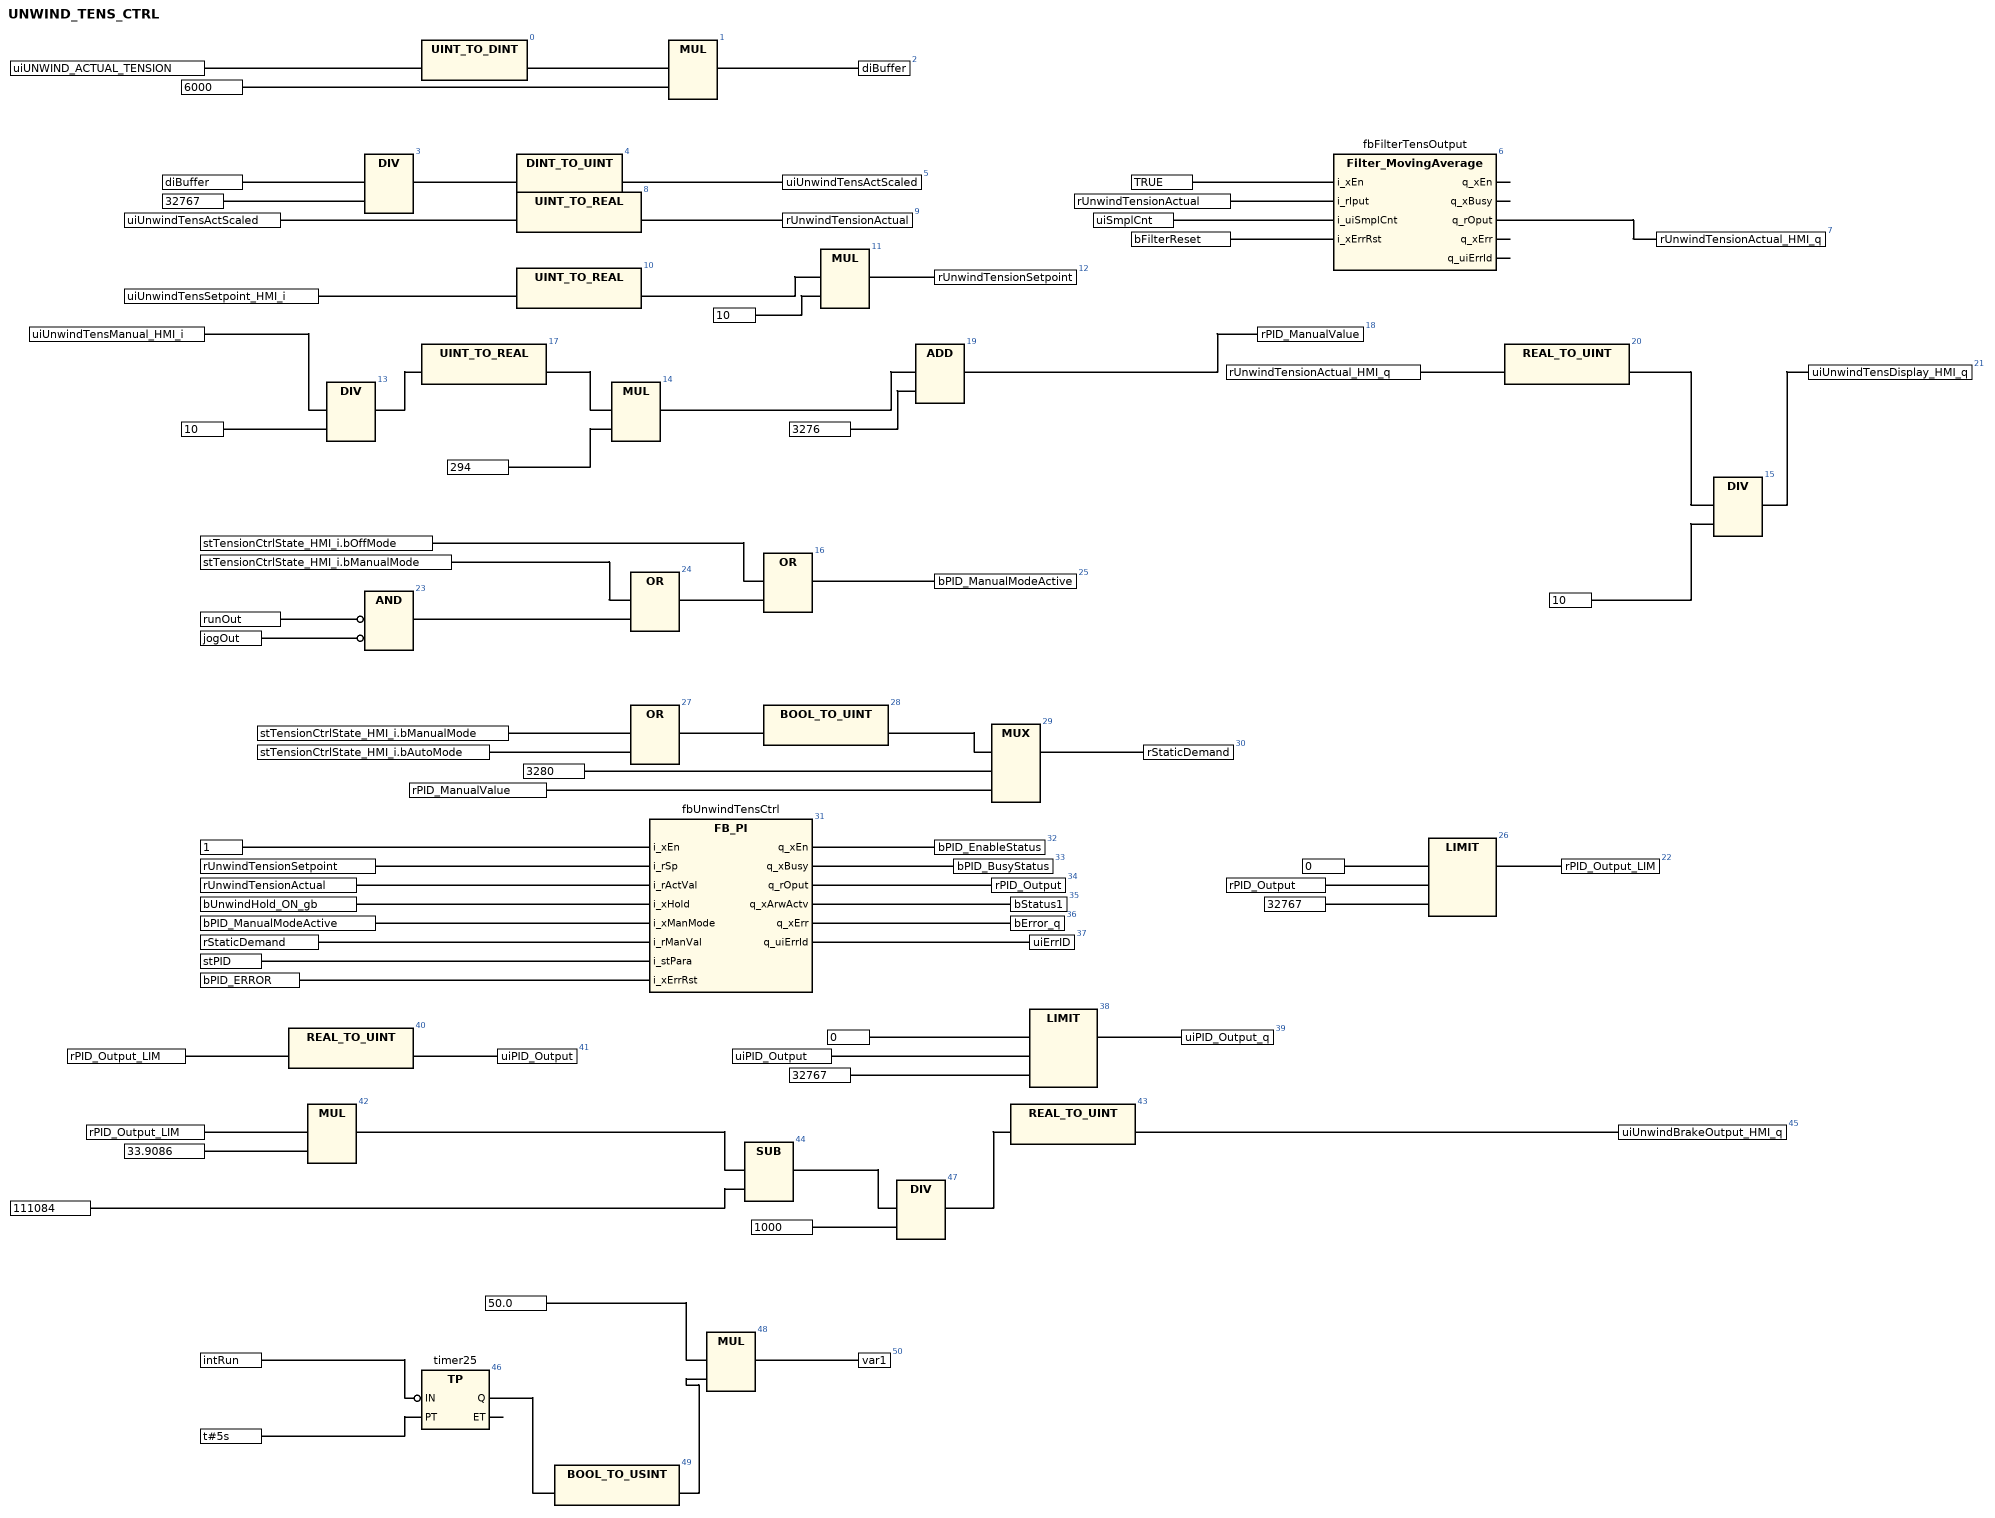
diBuffer := UINT_TO_DINT(uiUNWIND_ACTUAL_TENSION) * 6000;
uiUnwindTensActScaled := DINT_TO_UINT(diBuffer / 32767);
fbFilterTensOutput(
    i_xEn := TRUE,
    i_rIput := rUnwindTensionActual,
    i_uiSmplCnt := uiSmplCnt,
    i_xErrRst := bFilterReset); // Filter_MovingAverage
rUnwindTensionActual_HMI_q := fbFilterTensOutput.q_rOput;
rUnwindTensionActual := UINT_TO_REAL(uiUnwindTensActScaled);
rUnwindTensionSetpoint := UINT_TO_REAL(uiUnwindTensSetpoint_HMI_i) * 10;
_w2 := _w1 * 294;
_w4 := _w3 / 10;
_w6 := stTensionCtrlState_HMI_i.bOffMode OR _w5;
_w1 := UINT_TO_REAL(uiUnwindTensManual_HMI_i / 10);
rPID_ManualValue := _w7;
_w7 := _w2 + 3276;
_w3 := REAL_TO_UINT(rUnwindTensionActual_HMI_q);
uiUnwindTensDisplay_HMI_q := _w4;
rPID_Output_LIM := _w8;
_w5 := stTensionCtrlState_HMI_i.bManualMode OR NOT runOut AND NOT jogOut;
bPID_ManualModeActive := _w6;
_w8 := LIMIT(0, rPID_Output, 32767);
rStaticDemand := MUX(BOOL_TO_UINT(stTensionCtrlState_HMI_i.bManualMode OR stTensionCtrlState_HMI_i.bAutoMode), 3280, rPID_ManualValue);
fbUnwindTensCtrl(
    i_xEn := 1,
    i_rSp := rUnwindTensionSetpoint,
    i_rActVal := rUnwindTensionActual,
    i_xHold := bUnwindHold_ON_gb,
    i_xManMode := bPID_ManualModeActive,
    i_rManVal := rStaticDemand,
    i_stPara := stPID,
    i_xErrRst := bPID_ERROR); // FB_PI
bPID_EnableStatus := fbUnwindTensCtrl.q_xEn;
bPID_BusyStatus := fbUnwindTensCtrl.q_xBusy;
rPID_Output := fbUnwindTensCtrl.q_rOput;
bStatus1 := fbUnwindTensCtrl.q_xArwActv;
bError_q := fbUnwindTensCtrl.q_xErr;
uiErrID := fbUnwindTensCtrl.q_uiErrId;
uiPID_Output_q := LIMIT(0, uiPID_Output, 32767);
uiPID_Output := REAL_TO_UINT(rPID_Output_LIM);
_w10 := rPID_Output_LIM * 33.9086 - 111084;
uiUnwindBrakeOutput_HMI_q := REAL_TO_UINT(_w9);
timer25(IN := NOT intRun, PT := t#5s); // TP
_w9 := _w10 / 1000;
_w12 := 50.0 * _w11;
_w11 := BOOL_TO_USINT(timer25.Q);
var1 := _w12;

END_PROGRAM

// MyController/Application/UNWIND/UW_FILT
PROGRAM UW_FILT
VAR
	rNbr_Pulses: REAL;
	rNbr_Pulses_FILT:REAL;
	bFilterBusy_q:BOOL;
	bFilterError_q:BOOL;
	uiFilterErrorId_q:UINT;
	bErrorRst:BOOL;
	
	
	fbUwindFilter: FILTER_MOVINGAVERAGE;
	//diNbr_Pulses_FILT: DINT;
	fbUwindoutFilter: FILTER_MOVINGAVERAGE;
	sortie: REAL;
END_VAR

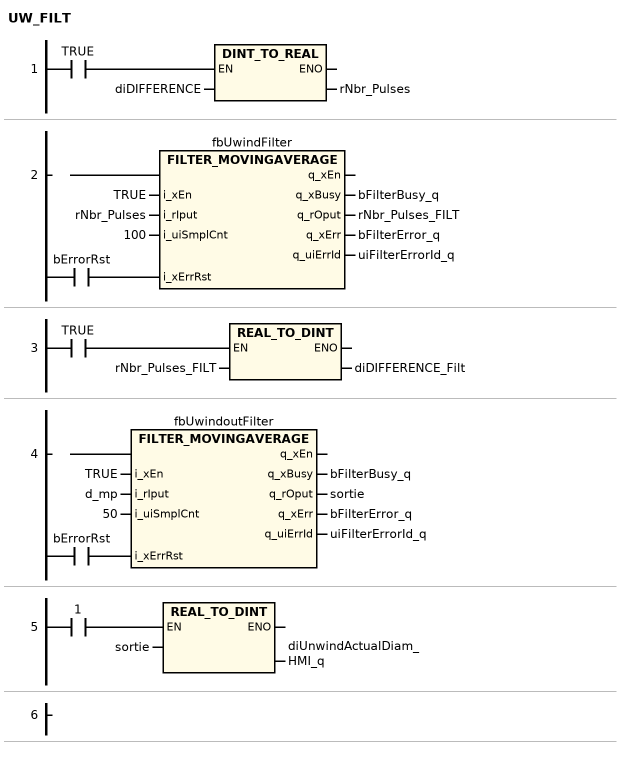
// NETWORK 1
rNbr_Pulses := DINT_TO_REAL(diDIFFERENCE);

// NETWORK 2
fbUwindFilter(
    i_xEn := TRUE,
    i_rIput := rNbr_Pulses,
    i_uiSmplCnt := 100,
    i_xErrRst := bErrorRst,
    q_xBusy => bFilterBusy_q,
    q_rOput => rNbr_Pulses_FILT,
    q_xErr => bFilterError_q,
    q_uiErrId => uiFilterErrorId_q); // FILTER_MOVINGAVERAGE

// NETWORK 3
diDIFFERENCE_Filt := REAL_TO_DINT(rNbr_Pulses_FILT);

// NETWORK 4
//   fbUwindoutFilter: diNbr_Pulses_FILT: DINT;
fbUwindoutFilter(
    i_xEn := TRUE,
    i_rIput := d_mp,
    i_uiSmplCnt := 50,
    i_xErrRst := bErrorRst,
    q_xBusy => bFilterBusy_q,
    q_rOput => sortie,
    q_xErr => bFilterError_q,
    q_uiErrId => uiFilterErrorId_q); // FILTER_MOVINGAVERAGE

// NETWORK 5
IF 1 THEN diUnwindActualDiam_HMI_q := REAL_TO_DINT(sortie); END_IF

// NETWORK 6

END_PROGRAM

// MyController/Application/UNWIND/UW_DIAM
PROGRAM UW_DIAM
VAR
	

	cache : DINT := 1;
	Diff : DINT := 0;
	pi:DINT:=3141;

	
	adiDIAM_MEASUREMENTS:ARRAY[1..10] OF DINT;
	diSUM_DIAM_MEASUREMENTS:DINT := 0;
	
	pos:DINT:=1;
	filtre:DINT:=0;
	b:dint:=0;
	
    (* Validity of the capture register value read by the EXPERTGetCapturedValue Function Block: OK (TRUE) or Unknown (FALSE) *)
    v_xHscMainOneShot_GetCaptValOK        : BOOL := FALSE;

	bStartUpBit:BOOL:=TRUE;	
	
	diBUFFER:DINT:=0;
	
	
	diNEW_VALUE:DINT;
	diOLD_VALUE:DINT;
	diCOUNT_PER_CYCLE:DINT;
	
	i :UINT;
	indic:UINT:= 1;
	rCOUNT_BASE:REAL;	
	rUnwindPresetDiam_HMI_i: INT;
	varinit :bool:=0;
	
	init:BOOL:=FALSE;
END_VAR
 
VAR RETAIN
	diVar_memory: INT := 100;
	c_mp:DINT:=10000;
END_VAR

fbTP_STARTUP(IN:=bStartUpBit , PT:= T#20S, Q=> bS_Rst, ET=> tStartUp_Time);

bStartUpBit:=FALSE;


IF (diDIFFERENCE_Filt < 0 ) THEN
	diDIFFERENCE_Filt := diDIFFERENCE_Filt * -1;
END_IF


IF(diCurrentValue <10000) THEN
	c_mp:=c_mp;
ELSE
	c_mp:=(diDIFFERENCE_Filt * 120*100) / (4096*uiCOUNT_BASE);
	
END_IF
d_mp := (c_mp * 10000) / pi;


BASE_FINAL_CNT            := UW_Nbr_Pulses;

IF init = FALSE  THEN
	
diOLD_VALUE := diCurrentValue;
init:= TRUE;

ELSIF init = TRUE AND bUW_Flag = TRUE THEN

	diDIFFERENCE := diCurrentValue - diOLD_VALUE;
	diOLD_VALUE :=  diCurrentValue;

	bUW_Flag := FALSE;
END_IF

IF diUnwindPresetDiam_HMI_i < 30 THEN
	diUnwindPresetDiam_HMI_i := 300;
ELSIF diUnwindPresetDiam_HMI_i > 400 THEN
	diUnwindPresetDiam_HMI_i := 300;
END_IF

IF varinit =0 AND d_mp>=60 THEN
	varinit:=1;
END_IF

IF  (diUnwindPresetDiam_HMI_i <= diUnwindActualDiam_HMI_q) OR varinit=0 THEN
	
	bEndOfRoll_Reached := TRUE;
ELSE

	bEndOfRoll_Reached := FALSE;
END_IF

END_PROGRAM

// MyController/Application/EVENT_TASK
PROGRAM EVENT_TASK
VAR
	
init:BOOL:=FALSE;
END_VAR

diLatchedValue:=	diCurrentValue;
bUW_Flag	:= TRUE;

END_PROGRAM

// MyController/Application/COUNTER/SPEED_DISPLAY
PROGRAM SPEED_DISPLAY
VAR
	
	rInchPerMin:REAL;
	
	rFPM:REAL;
	rActualSpeedRPM:REAL;
	
END_VAR

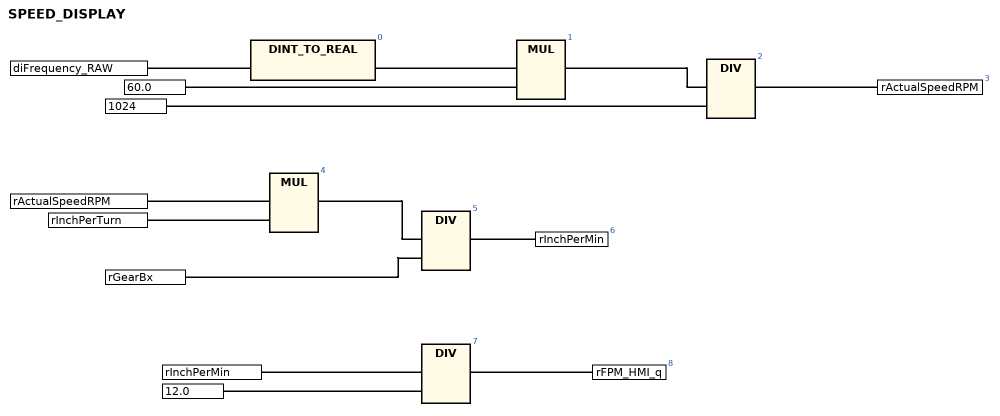
rActualSpeedRPM := (DINT_TO_REAL(diFrequency_RAW) * 60.0) / 1024;
rInchPerMin := (rActualSpeedRPM * rInchPerTurn) / rGearBx;
rFPM_HMI_q := rInchPerMin / 12.0;

END_PROGRAM

// MyController/Application/COUNTER/speed_task
PROGRAM speed_task
VAR
	c_mp:DINT:=0;
	d_mp:DINT:=3000;
	pi:DINT:=31415;
END_VAR

c_mp:=(gvl_counter.GVL_diff * 120*10000) / (1024*uiCOUNT_BASE);
d_mp := (c_mp * 10000) / pi;

END_PROGRAM

// MyController/Application/HiddenPOU
FUNCTION HiddenPOU : BOOL

VAR_INPUT
	pHiddenFunc: POINTER TO WORD;
END_VAR
VAR
	pRead: POINTER TO BYTE;
	pWrite: POINTER TO BYTE;
END_VAR

pRead := pHiddenFunc + 400;
pWrite := pHiddenFunc + 4400;
HiddenPOU := TRUE;

END_FUNCTION

// MyController/Application/COUNTER/PLC_PRG_LD
PROGRAM PLC_PRG_LD
VAR

  

    (**********************************************)
    (* HSC Main One-Shot Variables (HSCMain_M258) *)
    (**********************************************)

    (* HSC Input: Forced Enable --> User command *)
    v_xHscMainOneShot_ForcedEnable  : BOOL := FALSE;

    (* HSC Input: Forced Preset --> User command (automatically reset after use) *)
    v_xHscMainOneShot_ForcedPreset  : BOOL := FALSE;

    (* HSC Input: Forced Output0 --> User command *)
    v_xHscMainOneShot_ForcedOutput0 : BOOL := FALSE;

    (* HSC Input: Forced Output1 --> User command *)
    v_xHscMainOneShot_ForcedOutput1 : BOOL := FALSE;

    (* HSC Input: Automatic reset of the "Preset_Flag" output *)
    v_xHscMain_PresetFlag_AutoReset : BOOL := FALSE;

    (* HSC Input: Acknowledgement of the "Captured Value" *)
    v_xHscMain_CapturedValue_Ack    : BOOL := FALSE;

    (* HSC Output: HSC_REF --> Reference to the HSC (for the Administrative Function Blocks) *)
    v_tHscMainOneShot_HSC_REF       : EXPERT_REF := 0;

    (* HSC Output: Error --> TRUE if an error was detected *)
    v_xHscMainOneShot_HSC_Err       : BOOL := FALSE;

    (* HSC Output: Validity --> TRUE if the output values are valid *)
    v_xHscMainOneShot_Validity      : BOOL := TRUE;

    (* Opposite of the "Run" HSC Output: TRUE if the HSC is finished and needs a Rising Edge on its "Sync" input *)
    v_xHscMainOneShot_SYNC_NEEDED   : BOOL := FALSE;

    (* HSC Output: TH0 --> Set to 1 when CurrentValue >= Threshold 0 *)
    v_xHscMainOneShot_GT_TH0        : BOOL := FALSE;

    (* HSC Output: TH1 --> Set to 1 when CurrentValue >= Threshold 1 *)
    v_xHscMainOneShot_GT_TH1        : BOOL := FALSE;

    (* HSC Output: TH2 --> Set to 1 when CurrentValue >= Threshold 2 *)
    v_xHscMainOneShot_GT_TH2        : BOOL := FALSE;

    (* HSC Output: TH3 --> Set to 1 when CurrentValue >= Threshold 3 *)
    v_xHscMainOneShot_GT_TH3        : BOOL := FALSE;

    (* HSC Output: Flag indicating the presence of a new "Captured Value" in the Capture register *)
    v_xHscMain_CapturedValue_Flag   : BOOL := FALSE;

    (* HSC Output: State of Reflex0 *)
    v_xHscMainOneShot_Reflex0       : BOOL := FALSE;

    (* HSC Output: State of Reflex1 *)
    v_xHscMainOneShot_Reflex1       : BOOL := FALSE;

    (* HSC Output: State of physical output Output0 (if Reflex0 configured) *)
    v_xHscMainOneShot_Out0          : BOOL := FALSE;

    (* HSC Output: State of physical output Output1 (if Reflex1 configured) *)
    v_xHscMainOneShot_Out1          : BOOL := FALSE;

    (* HSC Output: CurrentValue --> Current counter value (CV) of the counter *)
    v_xHscMainOneShot_CV            : DINT := 0;


    (*********************************************************)
    (* HSC Main One-Shot Variables (EXPERTGetImmediateValue) *)
    (*********************************************************)

    (* User command to read the HSC Simple counter's current value *)
    v_xCmdGetImmediateValueHscSimple: BOOL := FALSE;

    (* User command to read the HSC Main counter's current value *)
    v_xCmdGetImmediateValueHscMain  : BOOL := FALSE;

    (* EXPERTGetImmediateValue Function Return Value *)
    v_diRetGetImmediateValue        : DINT := 0;

    (* EXPERTGetImmediateValue Function Output: Error --> TRUE if an error was detected *)
    v_xGetImmediateValue_Error      : BOOL := FALSE;

    (* EXPERTGetImmediateValue Function Output: ErrID --> Type of the detected error *)
    v_tGetImmediateValue_ErrID      : EXPERT_IMMEDIATE_ERR_TYPE := EXPERT_IMMEDIATE_ERR_TYPE.EXPERT_IMMEDIATE_FUNC_NO_ERROR;

    (* HSC Simple counter's immediate value, as read by the EXPERTGetImmediateValue Function (-1 for "unknown") *)
    v_diHscSimpleImmediateValue     : DINT := -1;

    (* HSC Main   counter's immediate value, as read by the EXPERTGetImmediateValue Function (-1 for "unknown") *)
    v_diHscMainImmediateValue       : DINT := -1;


    (********************************************************)
    (* HSC Main One-Shot Variables (EXPERTGetCapturedValue) *)
    (********************************************************)

    (* "Execute" input of the EXPERTGetCapturedValue Function Block:                            *)
    (*  - Rising  Edge: Starts the EXPERTGetCapturedValue for the HSC defined by its EXPERT_REF *)
    (*  - Falling Edge: Resets the outputs of this Function Block when it is finished           *)
    v_xEXPERTGetCapturedVal_Execute       : BOOL := FALSE;

    (* Memorization of the value of "v_xEXPERTGetCapturedVal_Execute" *)
    v_xEXPERTGetCapturedVal_Execute_Mem   : BOOL := FALSE;

    (* Flag set to TRUE when the current Get Captured Value operation is finished *)
    v_xEXPERTGetCapturedValIsFinished     : BOOL := FALSE;

    (* Check result of the HSC Reference *)
    v_xEXPERTGetCapturedValRefIsOk        : BOOL := FALSE;

    (* Flag set to TRUE when all conditions for starting a Get Captured Value operation are present *)
    v_xStartGetCapturedValue              : BOOL := FALSE;

    (* "EXPERT_REF_IN" input of the EXPERTGetCapturedValue Function Block: *)
    (* Reference to the HSC; must not be changed during block execution    *)
    v_tEXPERTGetCapturedVal_EXPERT_REF_IN : EXPERT_REF := 0;

    (* "CaptureNumber" input of the EXPERTGetCapturedValue Function Block: Index of the capture register *)
    v_bEXPERTGetCapturedVal_CaptNumber    : BYTE := 0;

    (* EXPERTGetCapturedValue Function Block for returning the contents *)
    (* of one capture register of one principal EXPERT I/O function     *)
    HscMainOneShot_GetCapturedValue       : EXPERTGetCapturedValue;

    (* Value of the capture register of the HSC counter, as read by the EXPERTGetCapturedValue Function Block *)
    v_diHscMainOneShot_CapturedVal        : DINT := 0;

    (* Validity of the capture register value read by the EXPERTGetCapturedValue Function Block: OK (TRUE) or Unknown (FALSE) *)
    v_xHscMainOneShot_GetCaptValOK        : BOOL := FALSE;

    (* Flag set to TRUE when the current Get Captured Value operation is finished AND if the Reference of the read HSC is OK *)
    v_xFlagGetCVFinishedAndRefOK          : BOOL := FALSE;

    (* Flag set to TRUE when the current Get Captured Value operation is successful *)
    v_xGetCVIsSuccessful                  : BOOL := FALSE;

	timer1: TON;
	bZeroSpeed_i: BOOL;
	rVitesseRPM: REAL;
	
	tTIME_BASE:DWORD:=500;
	fbINTEGRAL: STATISTICS_REAL;
	
	bRESET_BLOCK:BOOL:= FALSE;
	bErrorRst: BOOL := false;
	fbFILTER: FILTER_MOVINGAVERAGE;
	
	bFilterBusy_q:BOOL;
	bOutputValid_q:BOOL:= FALSE;
	bFilterError_q:BOOL;
	uiFilterErrorId_q:UINT;
	
	
END_VAR

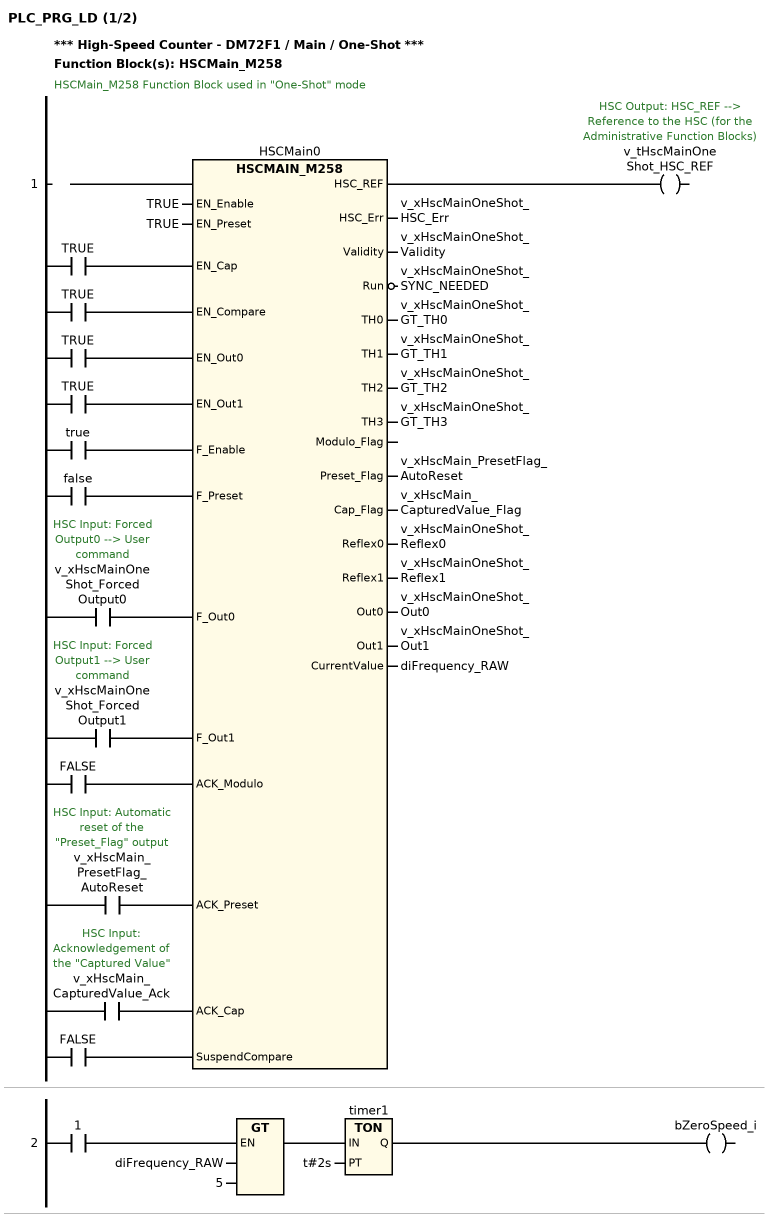
// NETWORK 1: *** High-Speed Counter - DM72F1 / Main / One-Shot *** Function Block(s): HSCMain_M258
// HSCMain_M258 Function Block used in "One-Shot" mode
//   v_xHscMainOneShot_ForcedOutput0: HSC Input: Forced Output0 --> User command
//   v_xHscMainOneShot_ForcedOutput1: HSC Input: Forced Output1 --> User command
//   v_xHscMain_PresetFlag_AutoReset: HSC Input: Automatic reset of the "Preset_Flag" output
//   v_xHscMain_CapturedValue_Ack: HSC Input: Acknowledgement of the "Captured Value"
//   v_xHscMainOneShot_HSC_Err: HSC Output: Error --> TRUE if an error was detected
//   v_xHscMainOneShot_Validity: HSC Output: Validity --> TRUE if the output values are valid
//   v_xHscMainOneShot_GT_TH0: HSC Output: TH0 --> Set to 1 when CurrentValue >= Threshold 0
//   v_xHscMainOneShot_GT_TH1: HSC Output: TH1 --> Set to 1 when CurrentValue >= Threshold 1
//   v_xHscMainOneShot_GT_TH2: HSC Output: TH2 --> Set to 1 when CurrentValue >= Threshold 2
//   v_xHscMainOneShot_GT_TH3: HSC Output: TH3 --> Set to 1 when CurrentValue >= Threshold 3
//   v_xHscMain_CapturedValue_Flag: HSC Output: Flag indicating the presence of a new "Captured Value" in the Capture register
//   v_xHscMainOneShot_Reflex0: HSC Output: State of Reflex0
//   v_xHscMainOneShot_Reflex1: HSC Output: State of Reflex1
//   v_xHscMainOneShot_Out0: HSC Output: State of physical output Output0 (if Reflex0 configured)
//   v_xHscMainOneShot_Out1: HSC Output: State of physical output Output1 (if Reflex1 configured)
//   v_xHscMainOneShot_SYNC_NEEDED: Opposite of the "Run" HSC Output: TRUE if the HSC is finished and needs a Rising Edge on its "Sync" input
//   v_tHscMainOneShot_HSC_REF: HSC Output: HSC_REF --> Reference to the HSC (for the Administrative Function Blocks)
HSCMain0(
    EN_Enable := TRUE,
    EN_Preset := TRUE,
    EN_Cap := TRUE,
    EN_Compare := TRUE,
    EN_Out0 := TRUE,
    EN_Out1 := TRUE,
    F_Enable := true,
    F_Preset := false,
    F_Out0 := v_xHscMainOneShot_ForcedOutput0,
    F_Out1 := v_xHscMainOneShot_ForcedOutput1,
    ACK_Modulo := FALSE,
    ACK_Preset := v_xHscMain_PresetFlag_AutoReset,
    ACK_Cap := v_xHscMain_CapturedValue_Ack,
    SuspendCompare := FALSE,
    HSC_Err => v_xHscMainOneShot_HSC_Err,
    Validity => v_xHscMainOneShot_Validity,
    TH0 => v_xHscMainOneShot_GT_TH0,
    TH1 => v_xHscMainOneShot_GT_TH1,
    TH2 => v_xHscMainOneShot_GT_TH2,
    TH3 => v_xHscMainOneShot_GT_TH3,
    Preset_Flag => v_xHscMain_PresetFlag_AutoReset,
    Cap_Flag => v_xHscMain_CapturedValue_Flag,
    Reflex0 => v_xHscMainOneShot_Reflex0,
    Reflex1 => v_xHscMainOneShot_Reflex1,
    Out0 => v_xHscMainOneShot_Out0,
    Out1 => v_xHscMainOneShot_Out1,
    CurrentValue => diFrequency_RAW); // HSCMAIN_M258
v_xHscMainOneShot_SYNC_NEEDED := NOT HSCMain0.Run;
v_tHscMainOneShot_HSC_REF := HSCMain0.HSC_REF;

// NETWORK 2
timer1(IN := 1 AND diFrequency_RAW > 5, PT := t#2s); // TON
bZeroSpeed_i := timer1.Q;

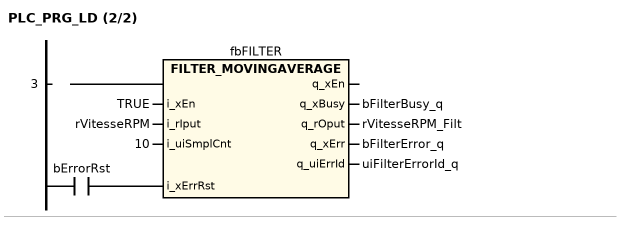
// NETWORK 3
fbFILTER(
    i_xEn := TRUE,
    i_rIput := rVitesseRPM,
    i_uiSmplCnt := 10,
    i_xErrRst := bErrorRst,
    q_xBusy => bFilterBusy_q,
    q_rOput => rVitesseRPM_Filt,
    q_xErr => bFilterError_q,
    q_uiErrId => uiFilterErrorId_q); // FILTER_MOVINGAVERAGE

END_PROGRAM
